(* CODESYS project BoxWrapper (3).project

Project tree, tasks and I/O mapping:
  Device : CODESYS Control Win V3 x64, 3S - Smart Software Solutions GmbH, version 3.5.12.20
    application Application
      libraries: Standard, * (System); VisuDialogs, * (System)
      task MainTask (cyclic, interval t#20ms, priority 1) calls BoxWrapperMain
      task VISU_TASK (cyclic, interval 100 ms, priority 31) calls VisuElems.Visu_Prg
      program PLC_PRG [LD]
      program BoxWrapperMain [LD]: Animation
      visualisation HMI
  text list GlobalTextList
*)

// Device/Application/BoxWrapperMain
PROGRAM BoxWrapperMain
VAR
	Start : BOOL;
	Stop  : BOOL;
	EMGC   : BOOL;
	RotationMotorCoil : BOOL;
	RotationMotorFreq : INT ;
	RotationMotorOVLD  : BOOL;
	
	SliderMotorUP			:BOOL;
	SliderMotorDown			:BOOL;
	SliderFreq				:INT;
	SliderOVLD				:BOOL;
	
	RotationCountPX			:BOOL;
	StretchPX				:BOOL;
	
	HLSW					:BOOL;
	LLSW					:BOOL;
	
	SliderLowCount			: CTU;
	SliderHighCount			:CTU;
	
 
 

 
	UpBlinker: TON;
	DownBlinker: TON;
	RotationBlinker: TON;
	UpDownCounterBlock: ctud;
	SliderCountValue: WORD;
	SliderCountAnimation: UINT;
	RotationCounterBlock: CTU;
	RotationCount: WORD;
 
	RotationFactor: INT;
	SliderFactor: INT;
END_VAR
VAR // added by the converter: edge detectors and wires of the graphical bodies
    _rt1, _rt2, _rt3, _rt4 : R_TRIG;
    _ft1 : F_TRIG;
END_VAR

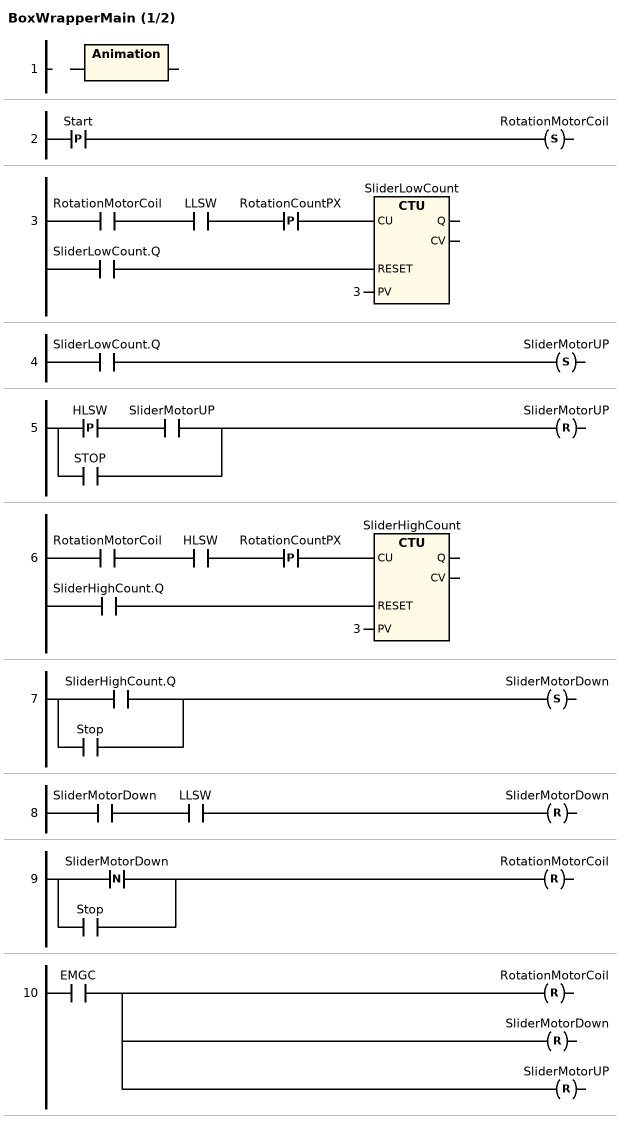
// NETWORK 1
Animation();

// NETWORK 2
_rt1(CLK := Start);
RotationMotorCoil S= _rt1.Q;

// NETWORK 3
_rt2(CLK := RotationCountPX);
SliderLowCount(CU := RotationMotorCoil AND LLSW AND _rt2.Q, RESET := SliderLowCount.Q, PV := 3); // CTU

// NETWORK 4
SliderMotorUP S= SliderLowCount.Q;

// NETWORK 5
_rt3(CLK := HLSW);
SliderMotorUP R= _rt3.Q AND SliderMotorUP OR STOP;

// NETWORK 6
_rt4(CLK := RotationCountPX);
SliderHighCount(CU := RotationMotorCoil AND HLSW AND _rt4.Q, RESET := SliderHighCount.Q, PV := 3); // CTU

// NETWORK 7
SliderMotorDown S= SliderHighCount.Q OR Stop;

// NETWORK 8
SliderMotorDown R= SliderMotorDown AND LLSW;

// NETWORK 9
_ft1(CLK := SliderMotorDown);
RotationMotorCoil R= _ft1.Q OR Stop;

// NETWORK 10
RotationMotorCoil R= EMGC;
SliderMotorDown R= EMGC;
SliderMotorUP R= EMGC;

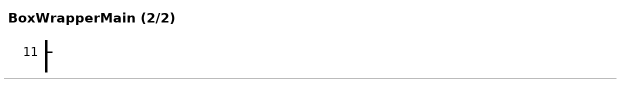
// NETWORK 11

ACTION Animation:
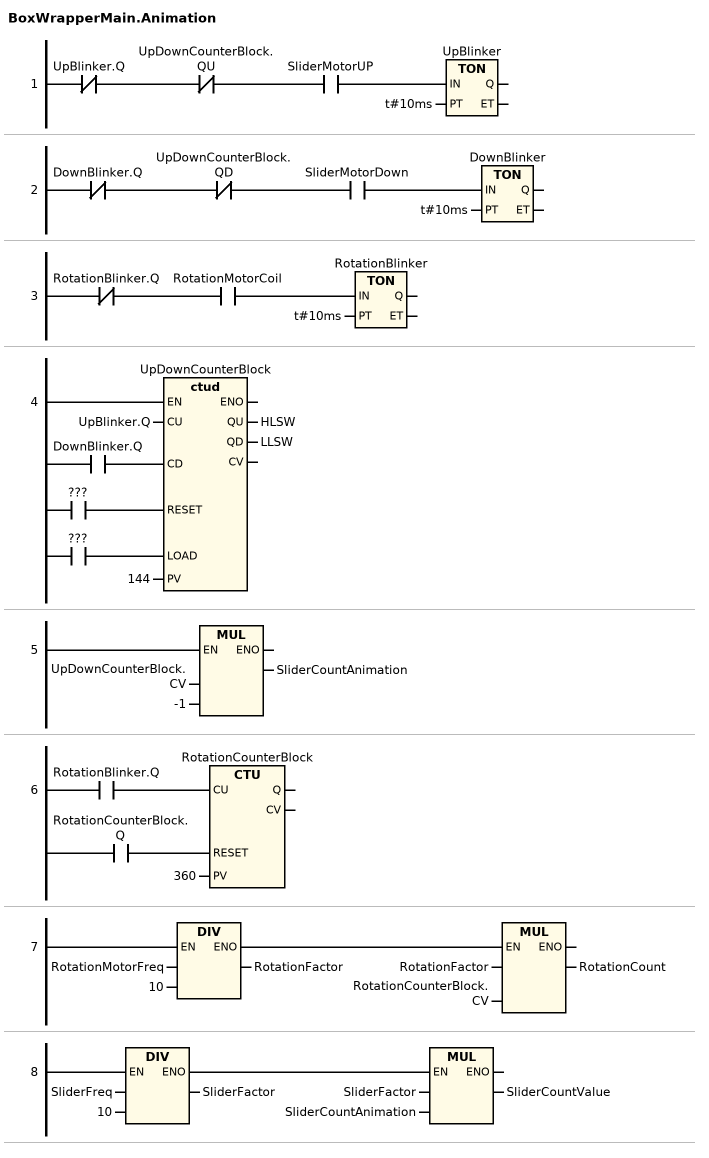
// NETWORK 1
UpBlinker(IN := NOT UpBlinker.Q AND NOT UpDownCounterBlock.QU AND SliderMotorUP, PT := t#10ms); // TON

// NETWORK 2
DownBlinker(IN := NOT DownBlinker.Q AND NOT UpDownCounterBlock.QD AND SliderMotorDown, PT := t#10ms); // TON

// NETWORK 3
RotationBlinker(IN := NOT RotationBlinker.Q AND RotationMotorCoil, PT := t#10ms); // TON

// NETWORK 4
UpDownCounterBlock(CU := UpBlinker.Q, CD := DownBlinker.Q, PV := 144, QU => HLSW, QD => LLSW); // ctud

// NETWORK 5
SliderCountAnimation := UpDownCounterBlock.CV * -1;

// NETWORK 6
RotationCounterBlock(CU := RotationBlinker.Q, RESET := RotationCounterBlock.Q, PV := 360); // CTU

// NETWORK 7
RotationFactor := RotationMotorFreq / 10;
RotationCount := RotationFactor * RotationCounterBlock.CV;

// NETWORK 8
SliderFactor := SliderFreq / 10;
SliderCountValue := SliderFactor * SliderCountAnimation;
END_ACTION

END_PROGRAM

// Device/Application/PLC_PRG
PROGRAM PLC_PRG
VAR
	Start : BOOL;
	Stop  : BOOL;
	RotationMotorCoil: BOOL;
	RotationMotorFreq:INT;
	RotationMotorOVLD:BOOL;
	Up_DownMotorCoil_UP : BOOL;
	Up_DownMotorCoil_DOWN : BOOL;
	Up_DownMotorFreq :INT;
	Up_DownMotorOVLD:BOOL;
	
	RotationCountProximity:BOOL;
	StretchWrap : BOOL;
	
	SW_Hi : BOOL;
	SW_Lw : BOOL;
	
	
	
	LowRotationCounter: CTU;
	HighRotationCounter: CTU;
END_VAR
VAR // added by the converter: edge detectors and wires of the graphical bodies
    _rt1, _rt2, _rt3, _rt4, _rt5, _rt6, _rt7 : R_TRIG;
    _ft1 : F_TRIG;
END_VAR

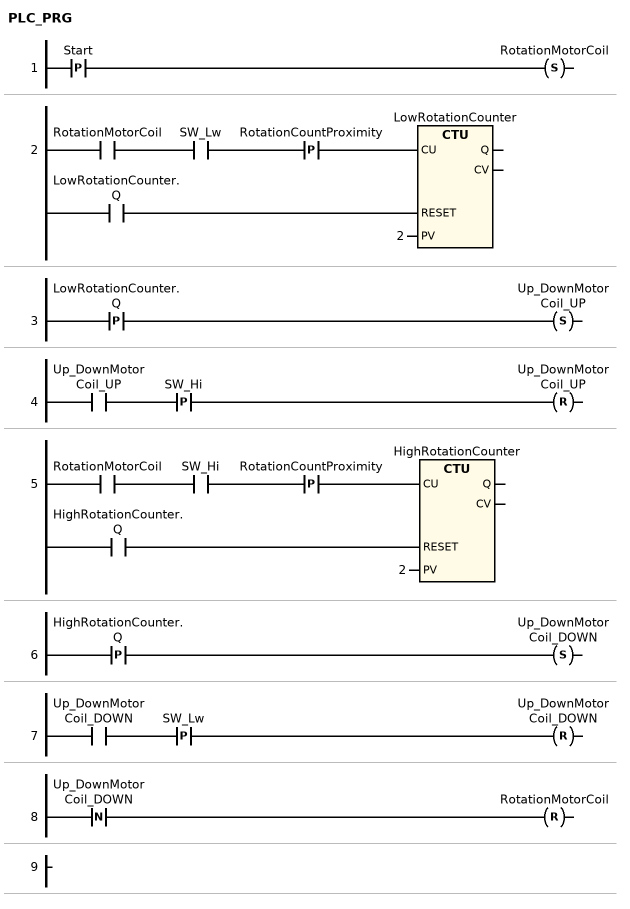
// NETWORK 1
_rt1(CLK := Start);
RotationMotorCoil S= _rt1.Q;

// NETWORK 2
_rt2(CLK := RotationCountProximity);
LowRotationCounter(CU := RotationMotorCoil AND SW_Lw AND _rt2.Q, RESET := LowRotationCounter.Q, PV := 2); // CTU

// NETWORK 3
_rt3(CLK := LowRotationCounter.Q);
Up_DownMotorCoil_UP S= _rt3.Q;

// NETWORK 4
_rt4(CLK := SW_Hi);
Up_DownMotorCoil_UP R= Up_DownMotorCoil_UP AND _rt4.Q;

// NETWORK 5
_rt5(CLK := RotationCountProximity);
HighRotationCounter(CU := RotationMotorCoil AND SW_Hi AND _rt5.Q, RESET := HighRotationCounter.Q, PV := 2); // CTU

// NETWORK 6
_rt6(CLK := HighRotationCounter.Q);
Up_DownMotorCoil_DOWN S= _rt6.Q;

// NETWORK 7
_rt7(CLK := SW_Lw);
Up_DownMotorCoil_DOWN R= Up_DownMotorCoil_DOWN AND _rt7.Q;

// NETWORK 8
_ft1(CLK := Up_DownMotorCoil_DOWN);
RotationMotorCoil R= _ft1.Q;

// NETWORK 9

END_PROGRAM

// Device/Application/HMI
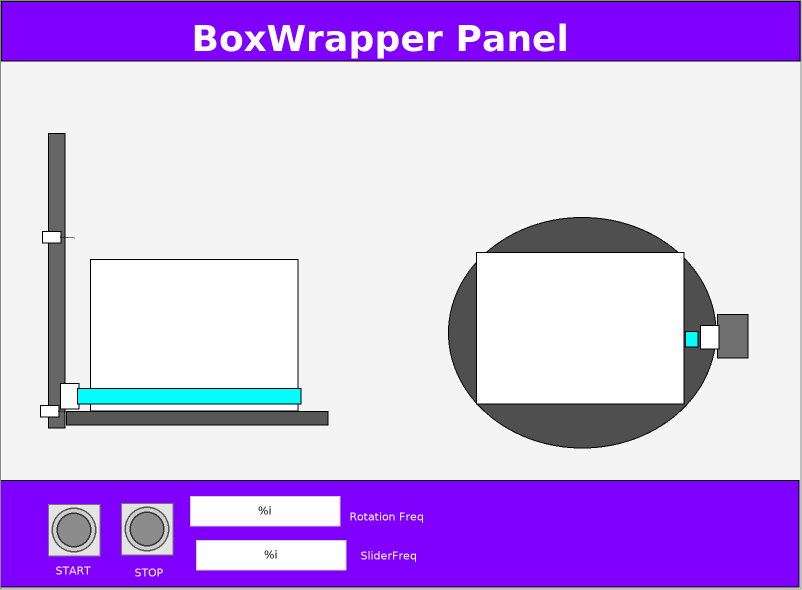
VISUALIZATION HMI  // 802x590
    Rectangle (1,1 799x60)
    Label (190,17 381x43), "BoxWrapper Panel"
    Rectangle (0,480 799x107)
    PushSwitch (120,503 54x52), variable: BoxWrapperMain.Stop, behaviour: TOGGLE, style: Switch-PushSwitch-Gray
    PushSwitch (47,504 54x52), variable: BoxWrapperMain.Start, behaviour: TOGGLE, style: Switch-PushSwitch-Gray
    Label (-2,556 150x30), "START"
    Label (74,558 150x30), "STOP"
    Label (314,541 150x30), "SliderFreq"
    Label (312,502 150x30), "Rotation Freq"
    Rectangle (48,133 17x295)
    RoundedRectangle (66,411 262x14)
    RoundedRectangle (90,259 208x152)
    Group (60,383 241x26)
        p2738717112: BoxWrapperMain.SliderCountAnimation
        RoundedRectangle (0,0 19x26)
        Rectangle (17,5 224x16)
    Group (42,231 32x12)
        RoundedRectangle (0,0 19x12)
        Line (32,7) (18,6)
    Group (40,405 32x12)
        RoundedRectangle (0,0 19x12)
        Line (32,7) (18,6)
    Ellipse (448,217 268x231)
    RoundedRectangle (476,252 208x152)
        p2858320360: BoxWrapperMain.RotationCount
    Rectangle (717,314 31x44)
    RoundedRectangle (700,325 19x24)
    Rectangle (685,331 13x16)
    Textfield (196,540 150x30), "%i", text variable: BoxWrapperMain.SliderFreq
        OnMouseClick: write the text variable via Default, min 0, max 50
    Textfield (190,496 150x30), "%i", text variable: BoxWrapperMain.RotationMotorFreq
        OnMouseClick: write the text variable via Default, min 0, max 50
END_VISUALIZATION
